TYPE
    ST_FeedInEmptyBox_Ctrl EXTENDS ST_CommandBasic :
    STRUCT
    END_STRUCT
END_TYPE

(* stored: Version 1.1.0.1, ProductVersion 3.1.4024.13
   DUT ST_FeedInEmptyBox_Ctrl: Id {fe3c0b16-bb39-4cfd-b130-a0e1a334512b} *)
